// TIA Portal V17 export
// export: Created 2024-08-07T21:44:00.9827316Z, ExportSetting WithDefaults, DisplayName Totally Integrated Automation Portal, DisplayVersion V17 Update 7, DisplayName TIA Portal Openness, DisplayVersion V17 Update 7, DisplayName TIA Portal Version Control Interface, DisplayVersion V17, DisplayName SINAMICS Startdrive Advanced, DisplayVersion V17 SP2, DisplayName SINAMICS Startdrive G110M, G120, G120C, G120D, G120P, G115D, DisplayVersion V17 SP2, DisplayName SINAMICS Startdrive G130, G150, S120, S150, SINAMICS MV, S210, DisplayVersion V17 SP2, DisplayName STEP 7 Professional, DisplayVersion V17 Update 7, DisplayName STEP 7 Safety, DisplayVersion V17 Update 6, DisplayName WinCC Advanced / Unified PC, DisplayVersion V17 Update 7
FUNCTION_BLOCK "Lamps"   // FB7, LAD
{ S7_Optimized_Access := 'TRUE' }
VERSION : 0.1
// stored: AutoNumber true, IsIECCheckEnabled false, IsRetainMemResEnabled false, MemoryReserve 100, SetENOAutomatically false, UDAEnableTagReadback false
   VAR
      R_TRIG_Instance { S7_SetPoint := 'True'} : R_TRIG;
      IEC_Timer_0_Instance { S7_SetPoint := 'True'} : TON_TIME;
   END_VAR
BEGIN

REGION Network 1: Lighthouse lamps
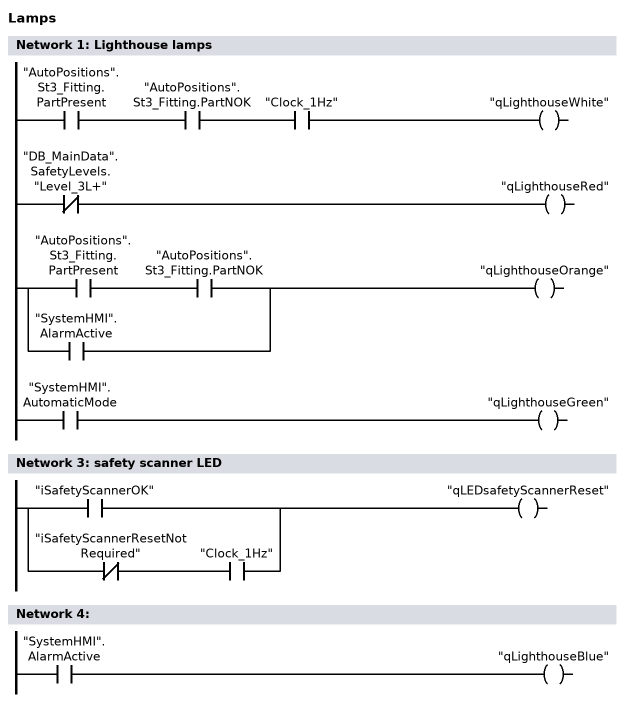
   RUNG wire#powerrail
      Contact( "AutoPositions".St3_Fitting.PartPresent )
      Contact( "AutoPositions".St3_Fitting.PartNOK )
      Contact( "Clock_1Hz" )
      Coil( "qLighthouseWhite" )
   END_RUNG
   RUNG wire#powerrail
      I_Contact( "DB_MainData".SafetyLevels."Level_3L+" )
      Coil( "qLighthouseRed" )
   END_RUNG
   RUNG wire#powerrail
      Contact( "AutoPositions".St3_Fitting.PartPresent )
      Contact( "AutoPositions".St3_Fitting.PartNOK )
      wire#w1
      Coil( "qLighthouseOrange" )
   END_RUNG
   RUNG wire#powerrail
      Contact( "SystemHMI".AlarmActive )
   END_RUNG wire#w1
   RUNG wire#powerrail
      Contact( "SystemHMI".AutomaticMode )
      Coil( "qLighthouseGreen" )
   END_RUNG
   // the same network as SCL:
   "qLighthouseWhite" := "AutoPositions".St3_Fitting.PartPresent AND "AutoPositions".St3_Fitting.PartNOK AND "Clock_1Hz";
   "qLighthouseRed" := NOT "DB_MainData".SafetyLevels."Level_3L+";
   "qLighthouseOrange" := ("AutoPositions".St3_Fitting.PartPresent AND "AutoPositions".St3_Fitting.PartNOK) OR "SystemHMI".AlarmActive;
   "qLighthouseGreen" := "SystemHMI".AutomaticMode;
END_REGION

REGION Network 2 (SCL): Alarm LED on OP
   //red button hmi
   "qResetAlarm" := "SystemHMI".AlarmActiveBlinking  AND "Clock_1Hz";
END_REGION

REGION Network 3: safety scanner LED
   RUNG wire#powerrail
      Contact( "iSafetyScannerOK" )
      wire#w1
      Coil( "qLEDsafetyScannerReset" )
   END_RUNG
   RUNG wire#powerrail
      I_Contact( "iSafetyScannerResetNotRequired" )
      Contact( "Clock_1Hz" )
   END_RUNG wire#w1
   // the same network as SCL:
   "qLEDsafetyScannerReset" := "iSafetyScannerOK" OR (NOT "iSafetyScannerResetNotRequired" AND "Clock_1Hz");
END_REGION

REGION Network 4
   RUNG wire#powerrail
      Contact( "SystemHMI".AlarmActive )
      Coil( "qLighthouseBlue" )
   END_RUNG
   // the same network as SCL:
   "qLighthouseBlue" := "SystemHMI".AlarmActive;
END_REGION
END_FUNCTION_BLOCK
